PROGRAM P_StackerBeltTable
VAR
		(*Initialization*)
	bSBT_OK		: BOOL;
	bError		: BOOL;
	bStart		: BOOL;
	bStop		: BOOL;
	(*Process*)
	bSBTEnable 	: BOOL;
	bSBTOn		: BOOL;
	bSBTOff		: BOOL;
	bOverride	: BOOL;
	//-----------------------------------------(*Case*)-----------------------------------------------------
	
	(* Reference for SBT

	State_Init 					,
	State_AutoStart         	,
	State_AutoStop          	,
	State_StackerStart			,
	State_StackerStop	        ,
	State_Override				,
	State_Error		

	*)	
	
END_VAR
VAR_INPUT
	bStartCommand : BOOL;
END_VAR
VAR_OUTPUT
	iSBTcase : INT;
END_VAR

CASE iSBTcase OF
StackerBeltTableState.State_Init			:
	IF bStartCommand 
	AND bSBT_OK 
	AND(NOT bError) THEN
		iSBTcase:=StackerBeltTableState.State_AutoStart;
	ELSE
		iSBTcase:=StackerBeltTableState.State_Error;
	END_IF 

StackerBeltTableState.State_AutoStart       :
	bSBTEnable	:= TRUE;
	iSBTcase	:= StackerBeltTableState.State_StackerStart;

StackerBeltTableState.State_AutoStop        :

StackerBeltTableState.State_StackerStart    : //Business Logic
	iSBTCase := StackerBeltTableState.State_Error;
	

StackerBeltTableState.State_StackerStop     : // Business Logic
	iSBTCase := StackerBeltTableState.State_Error;

StackerBeltTableState.State_Error           :
	IF (NOT bError) AND bSBTEnable THEN
		iSBTCase:=StackerBeltTableState.State_AutoStart;	
	END_IF
	IF bError THEN
		iSBTCase:=StackerBeltTableState.State_Init;	
	END_IF

StackerBeltTableState.State_Override        :
;

	
END_CASE

END_PROGRAM

(* stored: Version 1.1.0.1, ProductVersion 3.1.4024.12
   POU P_StackerBeltTable: Id {4d1169e7-1b8b-4f1c-bb90-5ea28424f6d7}, SpecialFunc None *)
